Fanuc TP program (LS listing): ground_truth.ls

/PROG  TOR_XL_LEARN_V4
/ATTR
OWNER		= MNEDITOR;
COMMENT		= "WeldPRO Auto-Gen";
PROG_SIZE	= 7125;
CREATE		= DATE 26-07-30  TIME 16:10:00;
MODIFIED	= DATE 26-07-30  TIME 16:41:22;
FILE_NAME	= TOR_XL_L;
VERSION		= 0;
LINE_COUNT	= 113;
MEMORY_SIZE	= 7445;
PROTECT		= READ_WRITE;
TCD:  STACK_SIZE	= 0,
      TASK_PRIORITY	= 50,
      TIME_SLICE	= 0,
      BUSY_LAMP_OFF	= 0,
      ABORT_REQUEST	= 0,
      PAUSE_REQUEST	= 0;
DEFAULT_GROUP	= 1,*,*,*,*;
CONTROL_CODE	= 00000000 00000000;
/APPL
/MN
   1:  !WeldPRO Auto-Generated TPP ;
   2:  !TOR_XL_2026, TOR_xl_2907 ;
   3:   ;
   4:  UFRAME_NUM=2 ;
   5:  UTOOL_NUM=2 ;
   6:  !Feature Approach ;
   7:J P[1]{
   GP1:
	UF : 2, UT : 2,		CONFIG : 'F D T, 0, 0, 0',
	X =   924.335  mm,	Y =   780.986  mm,	Z =  -268.284  mm,
	W =  -106.495 deg,	P =   -15.000 deg,	R =    94.234 deg
};
P[2]{
   GP1:
	UF : 2, UT : 2,		CONFIG : 'F D T, 0, 0, 0',
	X =  1018.649  mm,	Y =   786.723  mm,	Z =  -233.377  mm,
	W =  -106.492 deg,	P =   -15.098 deg,	R =    90.372 deg
};
P[3]{
   GP1:
	UF : 2, UT : 2,		CONFIG : 'F D T, 0, 0, 0',
	X =  1020.199  mm,	Y =   806.844  mm,	Z =  -233.327  mm,
	W =  -106.456 deg,	P =   -15.335 deg,	R =    80.815 deg
};
P[4]{
   GP1:
	UF : 2, UT : 2,		CONFIG : 'F D T, 0, 0, 0',
	X =  1022.000  mm,	Y =   816.895  mm,	Z =  -233.740  mm,
	W =  -106.423 deg,	P =   -15.450 deg,	R =    76.090 deg
};
P[5]{
   GP1:
	UF : 2, UT : 2,		CONFIG : 'F D T, 0, 0, 0',
	X =  1024.998  mm,	Y =   826.737  mm,	Z =  -234.474  mm,
	W =  -106.378 deg,	P =   -15.565 deg,	R =    71.217 deg
};
P[6]{
   GP1:
	UF : 2, UT : 2,		CONFIG : 'F D T, 0, 0, 0',
	X =  1028.901  mm,	Y =   836.094  mm,	Z =  -234.757  mm,
	W =  -106.322 deg,	P =   -15.679 deg,	R =    66.207 deg
};
P[7]{
   GP1:
	UF : 2, UT : 2,		CONFIG : 'F D T, 0, 0, 0',
	X =  1033.351  mm,	Y =   845.053  mm,	Z =  -234.666  mm,
	W =  -106.254 deg,	P =   -15.791 deg,	R =    61.015 deg
};
P[8]{
   GP1:
	UF : 2, UT : 2,		CONFIG : 'F D T, 0, 0, 0',
	X =  1038.941  mm,	Y =   853.294  mm,	Z =  -234.515  mm,
	W =  -106.177 deg,	P =   -15.894 deg,	R =    55.979 deg
};
P[9]{
   GP1:
	UF : 2, UT : 2,		CONFIG : 'F D T, 0, 0, 0',
	X =  1044.912  mm,	Y =   861.315  mm,	Z =  -234.681  mm,
	W =  -106.096 deg,	P =   -15.986 deg,	R =    51.162 deg
};
P[10]{
   GP1:
	UF : 2, UT : 2,		CONFIG : 'F D T, 0, 0, 0',
	X =  1051.319  mm,	Y =   869.011  mm,	Z =  -234.914  mm,
	W =  -106.012 deg,	P =   -16.066 deg,	R =    46.632 deg
};
P[11]{
   GP1:
	UF : 2, UT : 2,		CONFIG : 'F D T, 0, 0, 0',
	X =  1058.425  mm,	Y =   875.907  mm,	Z =  -234.815  mm,
	W =  -105.919 deg,	P =   -16.142 deg,	R =    41.952 deg
};
P[12]{
   GP1:
	UF : 2, UT : 2,		CONFIG : 'F D T, 0, 0, 0',
	X =  1066.038  mm,	Y =   882.624  mm,	Z =  -235.385  mm,
	W =  -105.870 deg,	P =   -16.177 deg,	R =    39.609 deg
};
P[13]{
   GP1:
	UF : 2, UT : 2,		CONFIG : 'F D T, 0, 0, 0',
	X =  1073.995  mm,	Y =   888.324  mm,	Z =  -234.902  mm,
	W =  -105.777 deg,	P =   -16.235 deg,	R =    35.365 deg
};
P[14]{
   GP1:
	UF : 2, UT : 2,		CONFIG : 'F D T, 0, 0, 0',
	X =  1082.325  mm,	Y =   893.929  mm,	Z =  -235.359  mm,
	W =  -105.677 deg,	P =   -16.289 deg,	R =    30.964 deg
};
P[15]{
   GP1:
	UF : 2, UT : 2,		CONFIG : 'F D T, 0, 0, 0',
	X =  1091.206  mm,	Y =   898.579  mm,	Z =  -235.754  mm,
	W =  -105.579 deg,	P =   -16.333 deg,	R =    26.830 deg
};
P[16]{
   GP1:
	UF : 2, UT : 2,		CONFIG : 'F D T, 0, 0, 0',
	X =  1100.054  mm,	Y =   902.724  mm,	Z =  -235.180  mm,
	W =  -105.537 deg,	P =   -16.344 deg,	R =    25.018 deg
};
P[17]{
   GP1:
	UF : 2, UT : 2,		CONFIG : 'F D T, 0, 0, 0',
	X =  1109.812  mm,	Y =   906.889  mm,	Z =  -236.313  mm,
	W =  -116.027 deg,	P =   -16.063 deg,	R =    30.267 deg
};
P[18]{
   GP1:
	UF : 2, UT : 2,		CONFIG : 'F D T, 0, 0, 0',
	X =  1118.461  mm,	Y =   911.370  mm,	Z =  -235.216  mm,
	W =  -126.877 deg,	P =   -15.356 deg,	R =    25.893 deg
};
P[19]{
   GP1:
	UF : 2, UT : 2,		CONFIG : 'F D T, 0, 0, 0',
	X =  1124.389  mm,	Y =   914.553  mm,	Z =  -229.472  mm,
	W =  -119.393 deg,	P =   -15.981 deg,	R =    16.221 deg
};
P[20]{
   GP1:
	UF : 2, UT : 2,		CONFIG : 'F D T, 0, 0, 0',
	X =  1130.108  mm,	Y =   917.570  mm,	Z =  -222.519  mm,
	W =  -115.329 deg,	P =   -16.208 deg,	R =    11.788 deg
};
P[21]{
   GP1:
	UF : 2, UT : 2,		CONFIG : 'F D T, 0, 0, 0',
	X =  1135.893  mm,	Y =   919.299  mm,	Z =  -214.215  mm,
	W =  -112.639 deg,	P =   -16.315 deg,	R =     9.714 deg
};
P[22]{
   GP1:
	UF : 2, UT : 2,		CONFIG : 'F D T, 0, 0, 0',
	X =  1142.785  mm,	Y =   921.790  mm,	Z =  -206.957  mm,
	W =  -110.015 deg,	P =   -16.386 deg,	R =     9.649 deg
};
P[23]{
   GP1:
	UF : 2, UT : 2,		CONFIG : 'F D T, 0, 0, 0',
	X =  1147.124  mm,	Y =   922.573  mm,	Z =  -202.837  mm,
	W =  -108.552 deg,	P =   -16.418 deg,	R =     8.950 deg
};
P[24]{
   GP1:
	UF : 2, UT : 2,		CONFIG : 'F D T, 0, 0, 0',
	X =  1160.405  mm,	Y =   924.073  mm,	Z =  -198.184  mm,
	W =  -105.409 deg,	P =   -16.443 deg,	R =     6.805 deg
};
P[25]{
   GP1:
	UF : 2, UT : 2,		CONFIG : 'F D T, 0, 0, 0',
	X =  1170.185  mm,	Y =   925.184  mm,	Z =  -197.751  mm,
	W =  -104.866 deg,	P =   -16.444 deg,	R =     5.597 deg
};
P[26]{
   GP1:
	UF : 2, UT : 2,		CONFIG : 'F D T, 0, 0, 0',
	X =  1179.875  mm,	Y =   926.246  mm,	Z =  -197.486  mm,
	W =  -104.887 deg,	P =   -16.444 deg,	R =     3.523 deg
};
P[27]{
   GP1:
	UF : 2, UT : 2,		CONFIG : 'F D T, 0, 0, 0',
	X =  1189.642  mm,	Y =   926.187  mm,	Z =  -197.840  mm,
	W =  -104.930 deg,	P =   -16.439 deg,	R =     -.729 deg
};
P[28]{
   GP1:
	UF : 2, UT : 2,		CONFIG : 'F D T, 0, 0, 0',
	X =  1199.192  mm,	Y =   925.409  mm,	Z =  -197.804  mm,
	W =  -104.979 deg,	P =   -16.424 deg,	R =    -5.541 deg
};
P[29]{
   GP1:
	UF : 2, UT : 2,		CONFIG : 'F D T, 0, 0, 0',
	X =  1208.963  mm,	Y =   924.598  mm,	Z =  -198.412  mm,
	W =  -105.028 deg,	P =   -16.400 deg,	R =   -10.259 deg
};
P[30]{
   GP1:
	UF : 2, UT : 2,		CONFIG : 'F D T, 0, 0, 0',
	X =  1218.399  mm,	Y =   922.765  mm,	Z =  -198.311  mm,
	W =  -105.070 deg,	P =   -16.371 deg,	R =   -14.490 deg
};
P[31]{
   GP1:
	UF : 2, UT : 2,		CONFIG : 'F D T, 0, 0, 0',
	X =  1228.031  mm,	Y =   920.244  mm,	Z =  -198.972  mm,
	W =  -105.112 deg,	P =   -16.334 deg,	R =   -18.515 deg
};
P[32]{
   GP1:
	UF : 2, UT : 2,		CONFIG : 'F D T, 0, 0, 0',
	X =  1237.147  mm,	Y =   916.829  mm,	Z =  -199.119  mm,
	W =  -105.158 deg,	P =   -16.285 deg,	R =   -23.051 deg
};
P[33]{
   GP1:
	UF : 2, UT : 2,		CONFIG : 'F D T, 0, 0, 0',
	X =  1245.892  mm,	Y =   912.712  mm,	Z =  -199.381  mm,
	W =  -105.219 deg,	P =   -16.204 deg,	R =   -29.417 deg
};
P[34]{
   GP1:
	UF : 2, UT : 2,		CONFIG : 'F D T, 0, 0, 0',
	X =  1253.810  mm,	Y =   907.751  mm,	Z =  -199.119  mm,
	W =  -105.311 deg,	P =   -16.047 deg,	R =   -39.415 deg
};
P[35]{
   GP1:
	UF : 2, UT : 2,		CONFIG : 'F D T, 0, 0, 0',
	X =  1261.433  mm,	Y =   901.277  mm,	Z =  -199.131  mm,
	W =  -105.307 deg,	P =   -16.055 deg,	R =   -38.974 deg
};
P[36]{
   GP1:
	UF : 2, UT : 2,		CONFIG : 'F D T, 0, 0, 0',
	X =  1269.012  mm,	Y =   894.754  mm,	Z =  -199.236  mm,
	W =  -105.302 deg,	P =   -16.063 deg,	R =   -38.625 deg
};
P[37]{
   GP1:
	UF : 2, UT : 2,		CONFIG : 'F D T, 0, 0, 0',
	X =  1277.147  mm,	Y =   889.161  mm,	Z =  -199.768  mm,
	W =  -105.469 deg,	P =   -15.944 deg,	R =   -44.976 deg
};
P[38]{
   GP1:
	UF : 2, UT : 2,		CONFIG : 'F D T, 0, 0, 0',
	X =  1283.666  mm,	Y =   882.089  mm,	Z =  -199.589  mm,
	W =  -105.661 deg,	P =   -15.890 deg,	R =   -47.714 deg
};
P[39]{
   GP1:
	UF : 2, UT : 2,		CONFIG : 'F D T, 0, 0, 0',
	X =  1290.668  mm,	Y =   875.216  mm,	Z =  -200.733  mm,
	W =  -106.210 deg,	P =   -15.792 deg,	R =   -52.259 deg
};
P[40]{
   GP1:
	UF : 2, UT : 2,		CONFIG : 'F D T, 0, 0, 0',
	X =  1295.955  mm,	Y =   867.182  mm,	Z =  -201.710  mm,
	W =  -106.927 deg,	P =   -15.688 deg,	R =   -56.663 deg
};
P[41]{
   GP1:
	UF : 2, UT : 2,		CONFIG : 'F D T, 0, 0, 0',
	X =  1302.253  mm,	Y =   859.600  mm,	Z =  -203.329  mm,
	W =  -107.603 deg,	P =   -15.597 deg,	R =   -60.243 deg
};
P[42]{
   GP1:
	UF : 2, UT : 2,		CONFIG : 'F D T, 0, 0, 0',
	X =  1307.276  mm,	Y =   851.059  mm,	Z =  -205.421  mm,
	W =  -108.271 deg,	P =   -15.504 deg,	R =   -63.685 deg
};
P[43]{
   GP1:
	UF : 2, UT : 2,		CONFIG : 'F D T, 0, 0, 0',
	X =  1311.178  mm,	Y =   842.174  mm,	Z =  -206.751  mm,
	W =  -109.144 deg,	P =   -15.377 deg,	R =   -68.203 deg
};
P[44]{
   GP1:
	UF : 2, UT : 2,		CONFIG : 'F D T, 0, 0, 0',
	X =  1315.606  mm,	Y =   833.024  mm,	Z =  -209.219  mm,
	W =  -109.899 deg,	P =   -15.253 deg,	R =   -72.505 deg
};
P[45]{
   GP1:
	UF : 2, UT : 2,		CONFIG : 'F D T, 0, 0, 0',
	X =  1318.210  mm,	Y =   823.515  mm,	Z =  -210.429  mm,
	W =  -110.273 deg,	P =   -15.181 deg,	R =   -74.981 deg
};
P[46]{
   GP1:
	UF : 2, UT : 2,		CONFIG : 'F D T, 0, 0, 0',
	X =  1320.230  mm,	Y =   813.739  mm,	Z =  -211.525  mm,
	W =  -110.635 deg,	P =   -14.305 deg,	R =   -78.232 deg
};
P[47]{
   GP1:
	UF : 2, UT : 2,		CONFIG : 'F D T, 0, 0, 0',
	X =  1321.758  mm,	Y =   803.727  mm,	Z =  -212.753  mm,
	W =  -111.054 deg,	P =   -14.769 deg,	R =   -83.164 deg
};
P[48]{
   GP1:
	UF : 2, UT : 2,		CONFIG : 'F D T, 0, 0, 0',
	X =  1322.258  mm,	Y =   793.690  mm,	Z =  -213.107  mm,
	W =  -111.190 deg,	P =   -15.305 deg,	R =   -88.308 deg
};
P[49]{
   GP1:
	UF : 2, UT : 2,		CONFIG : 'F D T, 0, 0, 0',
	X =  1322.489  mm,	Y =   783.619  mm,	Z =  -213.066  mm,
	W =  -111.129 deg,	P =   -15.645 deg,	R =   -91.614 deg
};
P[50]{
   GP1:
	UF : 2, UT : 2,		CONFIG : 'F D T, 0, 0, 0',
	X =  1322.436  mm,	Y =   773.380  mm,	Z =  -212.759  mm,
	W =  -110.761 deg,	P =   -14.624 deg,	R =   -96.574 deg
};
P[51]{
   GP1:
	UF : 2, UT : 2,		CONFIG : 'F D T, 0, 0, 0',
	X =  1320.760  mm,	Y =   763.539  mm,	Z =  -211.330  mm,
	W =  -110.276 deg,	P =   -14.535 deg,	R =  -100.836 deg
};
P[52]{
   GP1:
	UF : 2, UT : 2,		CONFIG : 'F D T, 0, 0, 0',
	X =  1319.036  mm,	Y =   753.689  mm,	Z =  -209.678  mm,
	W =  -109.635 deg,	P =   -14.447 deg,	R =  -105.265 deg
};
P[53]{
   GP1:
	UF : 2, UT : 2,		CONFIG : 'F D T, 0, 0, 0',
	X =  1316.263  mm,	Y =   744.113  mm,	Z =  -207.966  mm,
	W =  -109.083 deg,	P =   -14.382 deg,	R =  -108.625 deg
};
P[54]{
   GP1:
	UF : 2, UT : 2,		CONFIG : 'F D T, 0, 0, 0',
	X =  1312.685  mm,	Y =   734.730  mm,	Z =  -206.375  mm,
	W =  -108.349 deg,	P =   -14.302 deg,	R =  -112.873 deg
};
P[55]{
   GP1:
	UF : 2, UT : 2,		CONFIG : 'F D T, 0, 0, 0',
	X =  1309.141  mm,	Y =   725.309  mm,	Z =  -204.722  mm,
	W =  -107.748 deg,	P =   -14.239 deg,	R =  -116.265 deg
};
P[56]{
   GP1:
	UF : 2, UT : 2,		CONFIG : 'F D T, 0, 0, 0',
	X =  1304.757  mm,	Y =   716.421  mm,	Z =  -202.358  mm,
	W =  -106.927 deg,	P =   -14.148 deg,	R =  -121.193 deg
};
P[57]{
   GP1:
	UF : 2, UT : 2,		CONFIG : 'F D T, 0, 0, 0',
	X =  1299.321  mm,	Y =   707.941  mm,	Z =  -200.664  mm,
	W =  -106.269 deg,	P =   -14.066 deg,	R =  -125.698 deg
};
P[58]{
   GP1:
	UF : 2, UT : 2,		CONFIG : 'F D T, 0, 0, 0',
	X =  1292.959  mm,	Y =   700.183  mm,	Z =  -199.026  mm,
	W =  -105.781 deg,	P =   -13.988 deg,	R =  -130.143 deg
};
P[59]{
   GP1:
	UF : 2, UT : 2,		CONFIG : 'F D T, 0, 0, 0',
	X =  1286.719  mm,	Y =   692.361  mm,	Z =  -197.280  mm,
	W =  -105.527 deg,	P =   -13.913 deg,	R =  -134.519 deg
};
P[60]{
   GP1:
	UF : 2, UT : 2,		CONFIG : 'F D T, 0, 0, 0',
	X =  1279.894  mm,	Y =   684.848  mm,	Z =  -196.766  mm,
	W =  -105.437 deg,	P =   -13.849 deg,	R =  -138.629 deg
};
P[61]{
   GP1:
	UF : 2, UT : 2,		CONFIG : 'F D T, 0, 0, 0',
	X =  1272.475  mm,	Y =   678.006  mm,	Z =  -196.723  mm,
	W =  -105.429 deg,	P =   -13.831 deg,	R =  -139.837 deg
};
P[62]{
   GP1:
	UF : 2, UT : 2,		CONFIG : 'F D T, 0, 0, 0',
	X =  1265.641  mm,	Y =   670.880  mm,	Z =  -196.694  mm,
	W =  -105.443 deg,	P =   -13.863 deg,	R =  -137.727 deg
};
P[63]{
   GP1:
	UF : 2, UT : 2,		CONFIG : 'F D T, 0, 0, 0',
	X =  1257.021  mm,	Y =   664.482  mm,	Z =  -196.380  mm,
	W =  -105.373 deg,	P =   -13.729 deg,	R =  -147.436 deg
};
P[64]{
   GP1:
	UF : 2, UT : 2,		CONFIG : 'F D T, 0, 0, 0',
	X =  1247.675  mm,	Y =   659.504  mm,	Z =  -196.028  mm,
	W =  -105.298 deg,	P =   -13.637 deg,	R =  -156.529 deg
};
P[65]{
   GP1:
	UF : 2, UT : 2,		CONFIG : 'F D T, 0, 0, 0',
	X =  1238.718  mm,	Y =   654.671  mm,	Z =  -195.720  mm,
	W =  -105.277 deg,	P =   -13.618 deg,	R =  -158.976 deg
};
P[66]{
   GP1:
	UF : 2, UT : 2,		CONFIG : 'F D T, 0, 0, 0',
	X =  1229.140  mm,	Y =   650.755  mm,	Z =  -195.581  mm,
	W =  -105.241 deg,	P =   -13.592 deg,	R =  -162.969 deg
};
P[67]{
   GP1:
	UF : 2, UT : 2,		CONFIG : 'F D T, 0, 0, 0',
	X =  1219.150  mm,	Y =   648.586  mm,	Z =  -194.950  mm,
	W =  -105.203 deg,	P =   -13.573 deg,	R =  -167.022 deg
};
P[68]{
   GP1:
	UF : 2, UT : 2,		CONFIG : 'F D T, 0, 0, 0',
	X =  1208.995  mm,	Y =   646.891  mm,	Z =  -194.675  mm,
	W =  -105.159 deg,	P =   -13.560 deg,	R =  -171.569 deg
};
P[69]{
   GP1:
	UF : 2, UT : 2,		CONFIG : 'F D T, 0, 0, 0',
	X =  1198.788  mm,	Y =   645.638  mm,	Z =  -194.393  mm,
	W =  -105.113 deg,	P =   -13.556 deg,	R =  -176.312 deg
};
P[70]{
   GP1:
	UF : 2, UT : 2,		CONFIG : 'F D T, 0, 0, 0',
	X =  1188.607  mm,	Y =   645.777  mm,	Z =  -193.803  mm,
	W =  -105.068 deg,	P =   -13.561 deg,	R =   179.213 deg
};
P[71]{
   GP1:
	UF : 2, UT : 2,		CONFIG : 'F D T, 0, 0, 0',
	X =  1178.356  mm,	Y =   646.222  mm,	Z =  -194.041  mm,
	W =  -105.038 deg,	P =   -13.569 deg,	R =   176.231 deg
};
P[72]{
   GP1:
	UF : 2, UT : 2,		CONFIG : 'F D T, 0, 0, 0',
	X =  1168.405  mm,	Y =   646.885  mm,	Z =  -193.674  mm,
	W =  -105.207 deg,	P =   -13.572 deg,	R =   175.290 deg
};
P[73]{
   GP1:
	UF : 2, UT : 2,		CONFIG : 'F D T, 0, 0, 0',
	X =  1158.898  mm,	Y =   648.253  mm,	Z =  -194.274  mm,
	W =  -107.012 deg,	P =   -13.569 deg,	R =   174.537 deg
};
P[74]{
   GP1:
	UF : 2, UT : 2,		CONFIG : 'F D T, 0, 0, 0',
	X =  1150.196  mm,	Y =   649.161  mm,	Z =  -197.039  mm,
	W =  -109.414 deg,	P =   -13.538 deg,	R =   174.483 deg
};
P[75]{
   GP1:
	UF : 2, UT : 2,		CONFIG : 'F D T, 0, 0, 0',
	X =  1142.528  mm,	Y =   649.909  mm,	Z =  -202.837  mm,
	W =  -112.196 deg,	P =   -13.466 deg,	R =   175.323 deg
};
P[76]{
   GP1:
	UF : 2, UT : 2,		CONFIG : 'F D T, 0, 0, 0',
	X =  1136.214  mm,	Y =   650.722  mm,	Z =  -210.215  mm,
	W =  -114.872 deg,	P =   -13.369 deg,	R =   175.422 deg
};
P[77]{
   GP1:
	UF : 2, UT : 2,		CONFIG : 'F D T, 0, 0, 0',
	X =  1129.798  mm,	Y =   652.908  mm,	Z =  -217.766  mm,
	W =  -120.114 deg,	P =   -13.109 deg,	R =   172.293 deg
};
P[78]{
   GP1:
	UF : 2, UT : 2,		CONFIG : 'F D T, 0, 0, 0',
	X =  1123.352  mm,	Y =   657.737  mm,	Z =  -226.586  mm,
	W =  -126.810 deg,	P =   -12.622 deg,	R =   167.787 deg
};
P[79]{
   GP1:
	UF : 2, UT : 2,		CONFIG : 'F D T, 0, 0, 0',
	X =  1114.599  mm,	Y =   661.270  mm,	Z =  -230.856  mm,
	W =  -119.561 deg,	P =   -13.285 deg,	R =   157.806 deg
};
P[80]{
   GP1:
	UF : 2, UT : 2,		CONFIG : 'F D T, 0, 0, 0',
	X =  1105.442  mm,	Y =   665.774  mm,	Z =  -231.645  mm,
	W =  -107.219 deg,	P =   -13.741 deg,	R =   154.408 deg
};
P[81]{
   GP1:
	UF : 2, UT : 2,		CONFIG : 'F D T, 0, 0, 0',
	X =  1096.250  mm,	Y =   669.702  mm,	Z =  -231.594  mm,
	W =  -105.746 deg,	P =   -13.749 deg,	R =   154.142 deg
};
P[82]{
   GP1:
	UF : 2, UT : 2,		CONFIG : 'F D T, 0, 0, 0',
	X =  1087.130  mm,	Y =   674.159  mm,	Z =  -231.521  mm,
	W =  -105.804 deg,	P =   -13.784 deg,	R =   151.506 deg
};
P[83]{
   GP1:
	UF : 2, UT : 2,		CONFIG : 'F D T, 0, 0, 0',
	X =  1078.244  mm,	Y =   679.402  mm,	Z =  -231.746  mm,
	W =  -105.885 deg,	P =   -13.838 deg,	R =   147.739 deg
};
P[84]{
   GP1:
	UF : 2, UT : 2,		CONFIG : 'F D T, 0, 0, 0',
	X =  1069.572  mm,	Y =   685.221  mm,	Z =  -232.068  mm,
	W =  -105.988 deg,	P =   -13.918 deg,	R =   142.681 deg
};
P[85]{
   GP1:
	UF : 2, UT : 2,		CONFIG : 'F D T, 0, 0, 0',
	X =  1062.045  mm,	Y =   692.371  mm,	Z =  -232.268  mm,
	W =  -106.082 deg,	P =   -14.006 deg,	R =   137.688 deg
};
P[86]{
   GP1:
	UF : 2, UT : 2,		CONFIG : 'F D T, 0, 0, 0',
	X =  1054.613  mm,	Y =   699.088  mm,	Z =  -231.837  mm,
	W =  -106.129 deg,	P =   -14.056 deg,	R =   135.015 deg
};
P[87]{
   GP1:
	UF : 2, UT : 2,		CONFIG : 'F D T, 0, 0, 0',
	X =  1047.673  mm,	Y =   706.571  mm,	Z =  -231.870  mm,
	W =  -106.186 deg,	P =   -14.117 deg,	R =   131.622 deg
};
P[88]{
   GP1:
	UF : 2, UT : 2,		CONFIG : 'F D T, 0, 0, 0',
	X =  1041.440  mm,	Y =   714.732  mm,	Z =  -231.977  mm,
	W =  -106.269 deg,	P =   -14.239 deg,	R =   125.999 deg
};
P[89]{
   GP1:
	UF : 2, UT : 2,		CONFIG : 'F D T, 0, 0, 0',
	X =  1035.280  mm,	Y =   722.998  mm,	Z =  -232.670  mm,
	W =  -106.343 deg,	P =   -14.367 deg,	R =   120.225 deg
};
P[90]{
   GP1:
	UF : 2, UT : 2,		CONFIG : 'F D T, 0, 0, 0',
	X =  1030.835  mm,	Y =   732.218  mm,	Z =  -232.234  mm,
	W =  -106.384 deg,	P =   -14.458 deg,	R =   116.261 deg
};
P[91]{
   GP1:
	UF : 2, UT : 2,		CONFIG : 'F D T, 0, 0, 0',
	X =  1027.572  mm,	Y =   739.660  mm,	Z =  -232.418  mm,
	W =  -106.433 deg,	P =   -14.556 deg,	R =   111.957 deg
};
P[92]{
   GP1:
	UF : 2, UT : 2,		CONFIG : 'F D T, 0, 0, 0',
	X =  1023.534  mm,	Y =   751.390  mm,	Z =  -232.797  mm,
	W =  -106.465 deg,	P =   -14.714 deg,	R =   105.666 deg
};
P[93]{
   GP1:
	UF : 2, UT : 2,		CONFIG : 'F D T, 0, 1, 0',
	X =  1021.563  mm,	Y =   761.346  mm,	Z =  -232.974  mm,
	W =  -106.480 deg,	P =   -14.798 deg,	R =   102.262 deg
};
P[94]{
   GP1:
	UF : 2, UT : 2,		CONFIG : 'F D T, 0, 1, 0',
	X =  1019.328  mm,	Y =   771.303  mm,	Z =  -233.119  mm,
	W =  -106.494 deg,	P =   -14.935 deg,	R =    96.827 deg
};
P[95]{
   GP1:
	UF : 2, UT : 2,		CONFIG : 'F D T, 0, 1, 0',
	X =  1019.013  mm,	Y =   778.603  mm,	Z =  -233.253  mm,
	W =  -106.501 deg,	P =   -14.999 deg,	R =    94.236 deg
};
P[96]{
   GP1:
	UF : 2, UT : 2,		CONFIG : 'F D T, 0, 0, 0',
	X =  1018.962  mm,	Y =   778.590  mm,	Z =  -233.220  mm,
	W =  -106.499 deg,	P =   -14.997 deg,	R =    94.226 deg
};
P[97]{
   GP1:
	UF : 2, UT : 2,		CONFIG : 'F D T, 0, 0, 0',
	X =  1018.769  mm,	Y =   796.897  mm,	Z =  -233.531  mm,
	W =  -106.481 deg,	P =   -15.218 deg,	R =    85.605 deg
};
P[98]{
   GP1:
	UF : 2, UT : 2,		CONFIG : 'F D T, 0, 1, 0',
	X =   651.995  mm,	Y =   781.694  mm,	Z =  -345.952  mm,
	W =  -106.495 deg,	P =   -15.000 deg,	R =    94.234 deg
};

/END
